FUNCTION_BLOCK FB_Bel_Monitoring (* Baustein dient dem Monitoring einzelner Lampen bei Lampengruppen, d.h. insbesondere der Hallenbeleuchtung *)
VAR_INPUT
	Settings_Array	: ARRAY [0..63] OF ST_DALIV2DeviceSettings;
	Zustand			: ST_Bel_Zustand;
END_VAR
VAR_OUTPUT
END_VAR
VAR
	i	: INT;
	Relative_Leistung	: REAL;
END_VAR

FOR i := 0 TO 30 DO
	Zustand.Lampen_Monitoring[i].Betrieb := Settings_Array[i].bPresent;
	Relative_Leistung := Settings_Array[i].nActualLevel;
	Zustand.Lampen_Monitoring[i].Relative_Leistung := (Relative_Leistung - 126)/ 1.28;
END_FOR

END_FUNCTION_BLOCK

(* stored: Version 1.1.0.1, ProductVersion 3.1.4024.10
   POU FB_Bel_Monitoring: Id {8baaa502-b25f-4e5a-ad0b-69c450862fdf}, SpecialFunc None *)
